% RSLogix 500 project I2P JOB 13 - FORWARD-REVERSE USING 3 PBS OF 1P MOTOR.RSS, saved by version 10.00.00.00 %
PROJECT "ML5B"    % processor: Bul.1763 MicroLogix 1100 Series B %

PROGRAM FILES
  LAD 2   6 rungs

DATA FILES
  O0 OUTPUT  4 elements
  I1 INPUT  6 elements
  S2 STATUS  66 elements
  B3 BINARY  1 elements
  T4 TIMER  1 elements
  C5 COUNTER  1 elements
  R6 CONTROL  1 elements
  N7 INTEGER  1 elements
  F8 FLOAT  1 elements

LADDER 2
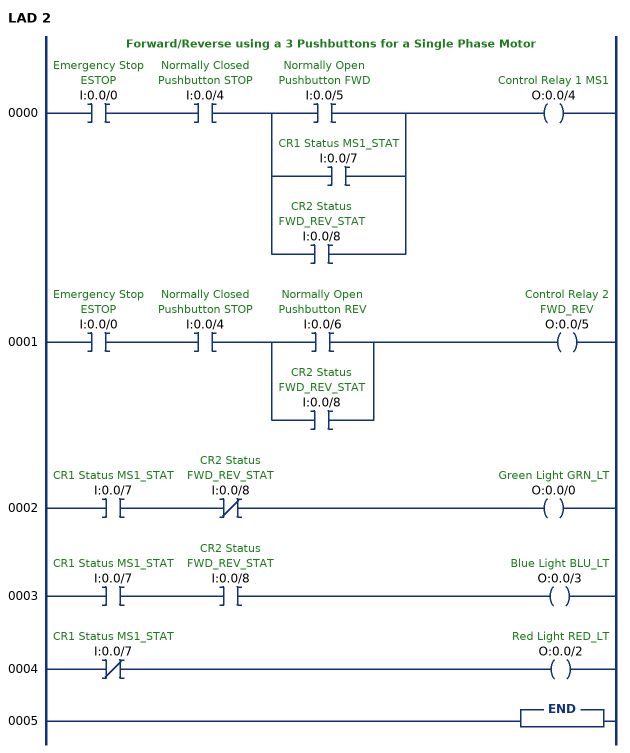
% Rung: 0 %
% TITLE: Forward/Reverse using a 3 Pushbuttons for a Single Phase Motor %
SOR XIC I:0.0/0 XIC I:0.0/4 BST XIC I:0.0/5 NXB XIC I:0.0/7 NXB XIC I:0.0/8 BND OTE O:0.0/4 EOR
%   I:0.0/0  ESTOP  "Emergency Stop" %
%   I:0.0/4  STOP  "Normally Closed Pushbutton" %
%   I:0.0/5  FWD  "Normally Open Pushbutton" %
%   I:0.0/7  MS1_STAT  "CR1 Status" %
%   I:0.0/8  FWD_REV_STAT  "CR2 Status" %
%   O:0.0/4  MS1  "Control Relay 1" %
% Rung: 1 %
SOR XIC I:0.0/0 XIC I:0.0/4 BST XIC I:0.0/6 NXB XIC I:0.0/8 BND OTE O:0.0/5 EOR
%   I:0.0/0  ESTOP  "Emergency Stop" %
%   I:0.0/4  STOP  "Normally Closed Pushbutton" %
%   I:0.0/6  REV  "Normally Open Pushbutton" %
%   I:0.0/8  FWD_REV_STAT  "CR2 Status" %
%   O:0.0/5  FWD_REV  "Control Relay 2" %
% Rung: 2 %
SOR XIC I:0.0/7 XIO I:0.0/8 OTE O:0.0/0 EOR
%   I:0.0/7  MS1_STAT  "CR1 Status" %
%   I:0.0/8  FWD_REV_STAT  "CR2 Status" %
%   O:0.0/0  GRN_LT  "Green Light" %
% Rung: 3 %
SOR XIC I:0.0/7 XIC I:0.0/8 OTE O:0.0/3 EOR
%   I:0.0/7  MS1_STAT  "CR1 Status" %
%   I:0.0/8  FWD_REV_STAT  "CR2 Status" %
%   O:0.0/3  BLU_LT  "Blue Light" %
% Rung: 4 %
SOR XIO I:0.0/7 OTE O:0.0/2 EOR
%   I:0.0/7  MS1_STAT  "CR1 Status" %
%   O:0.0/2  RED_LT  "Red Light" %
% Rung: 5 %
SOR END EOR

OTHER DOCUMENTED ADDRESSES
  I:0.0/1  3PSSA  "3 Position SS A"
  I:0.0/2  3PSSB  "3 Position SS B"
  I:0.0/3  2PSS  "2 Position SS"
  O:0.0/1  YLW_LT  "Yellow Light"
